// TIA Portal V20 export
TYPE "LER_typeCommunicationInterface"
// stored: Access Published
   STRUCT
      commands : "LER_typeCommunicationCommands";
      monitoring : "LER_typeCommunicationMonitoring";
      configuration : "LER_typeCommunicationConfiguration";
   END_STRUCT;
END_TYPE
